FUNCTION_BLOCK CROSSCOMM_SENDER_153F5A08CC8D75AF0 (* Service Interface Function Block Type *)
  (* Standard: 61499-2 *)
  (* Version 0.0, 9/22/2017, bababen, nxtControl GmbH, template *)
  PACKAGE Main;
  (* Compiler Cpp nxtControl builtin 1.0 *)
  {SET_ATTRIBUTE(Runtime.FBType.ImplementingType, Runtime.System#DYNGEN_CROSSCOMM_SENDER)}
  {SET_ATTRIBUTE(Configuration.GenericFBType.InterfaceParams, Runtime.System#<InterfaceList> <EventInputs> <Event Name="CNF"> <With Var="OUT" /> </Event> </EventInputs> <InputVars> <VarDeclaration Name="OUT" Type="TIME" /> </InputVars> </InterfaceList>)}
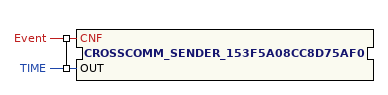
  EVENT_INPUT
    CNF WITH OUT;
  END_EVENT
  VAR_INPUT
    OUT : TIME;
  END_VAR
  EC_STATES
    START;
  END_STATES
END_FUNCTION_BLOCK
